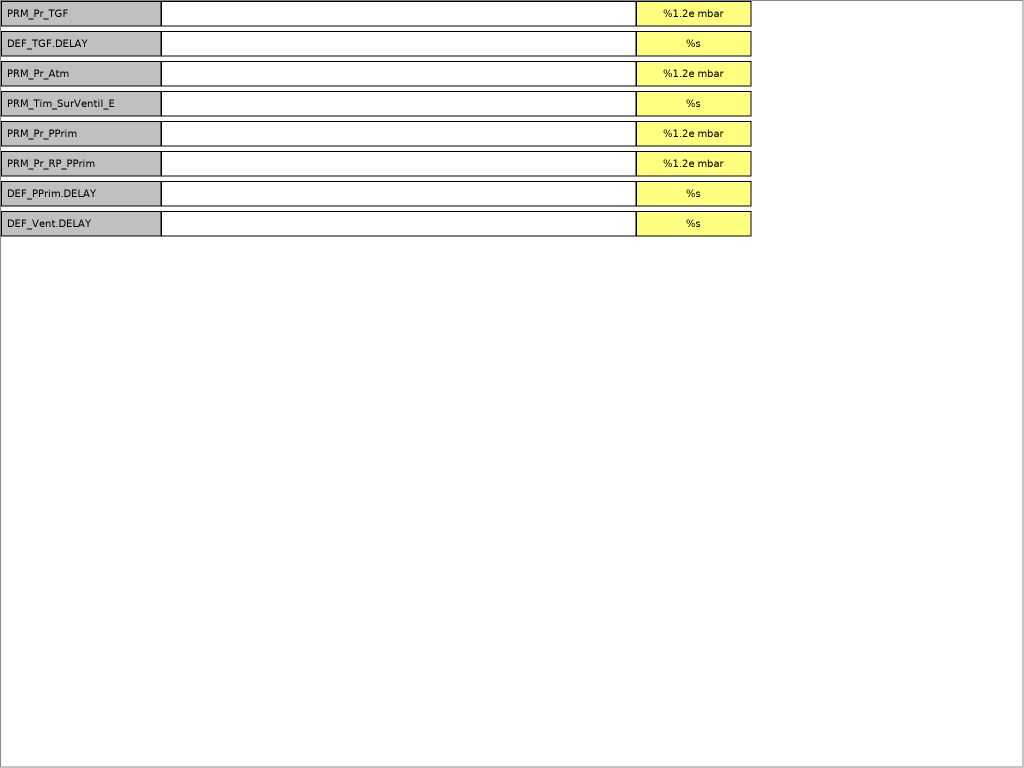
VISUALIZATION VISU_CONFIG_POMPAGE_SAS  // 1024x768
VAR_IN_OUT
	m_Input_PRG_POMPAGE : BLOCK_PRG_POMPAGE_SAS;
END_VAR
    Rectangle (161,1 475x25), text list: 'TextList_Config_Pompage', text index: 2
    Rectangle (636,1 115x25), "%1.2e mbar", text variable: m_Input_PRG_POMPAGE.POMPAGE.PRM_Pr_TGF, input disabled if: NOT Global_Variables.PRG_USER.ACTU_USER.CONF_MACHINE
        OnMouseClick: write the text variable via VisuDialogs.NumpadExtended, min 10, max 1000
    Rectangle (1,1 160x25), "PRM_Pr_TGF"
    Rectangle (161,31 475x25), text list: 'TextList_Config_Pompage', text index: 3
    Rectangle (636,31 115x25), "%s", text variable: m_Input_PRG_POMPAGE.POMPAGE.DEF_TGF.DELAY, input disabled if: NOT Global_Variables.PRG_USER.ACTU_USER.CONF_MACHINE
        OnMouseClick: write the text variable via VisuDialogs.Keypad
    Rectangle (1,31 160x25), "DEF_TGF.DELAY"
    Rectangle (161,61 475x25), text list: 'TextList_Config_Pompage', text index: 4
    Rectangle (161,91 475x25), text list: 'TextList_Config_Pompage', text index: 5
    Rectangle (636,61 115x25), "%1.2e mbar", text variable: m_Input_PRG_POMPAGE.POMPAGE.PRM_Pr_Atm, input disabled if: NOT Global_Variables.PRG_USER.ACTU_USER.CONF_MACHINE
        OnMouseClick: write the text variable via VisuDialogs.Numpad, min 100, max 1000
    Rectangle (1,61 160x25), "PRM_Pr_Atm"
    Rectangle (636,91 115x25), "%s", text variable: m_Input_PRG_POMPAGE.POMPAGE.PRM_Tim_SurVentil_E, input disabled if: NOT Global_Variables.PRG_USER.ACTU_USER.CONF_MACHINE
        OnMouseClick: write the text variable via VisuDialogs.Keypad
    Rectangle (1,91 160x25), "PRM_Tim_SurVentil_E"
    Rectangle (161,121 475x25), text list: 'TextList_Config_Pompage', text index: 6
    Rectangle (636,121 115x25), "%1.2e mbar", text variable: m_Input_PRG_POMPAGE.POMPAGE.PRM_Pr_PPrim, input disabled if: NOT Global_Variables.PRG_USER.ACTU_USER.CONF_MACHINE
        OnMouseClick: write the text variable via VisuDialogs.NumpadExtended, min 1e-3, max 1e-1
    Rectangle (1,121 160x25), "PRM_Pr_PPrim"
    Rectangle (1,151 160x25), "PRM_Pr_RP_PPrim"
    Rectangle (161,151 475x25), text list: 'TextList_Config_Pompage', text index: 7
    Rectangle (636,151 115x25), "%1.2e mbar", text variable: m_Input_PRG_POMPAGE.POMPAGE.PRM_Pr_RP_PPrim, input disabled if: NOT Global_Variables.PRG_USER.ACTU_USER.CONF_MACHINE
        OnMouseClick: write the text variable via VisuDialogs.NumpadExtended, min 1e-3, max 1e-1
    Rectangle (1,181 160x25), "DEF_PPrim.DELAY"
    Rectangle (161,181 475x25), text list: 'TextList_Config_Pompage', text index: 8
    Rectangle (636,181 115x25), "%s", text variable: m_Input_PRG_POMPAGE.POMPAGE.DEF_PPRIM.DELAY, input disabled if: NOT Global_Variables.PRG_USER.ACTU_USER.CONF_MACHINE
        OnMouseClick: write the text variable via VisuDialogs.Keypad
    Rectangle (1,211 160x25), "DEF_Vent.DELAY"
    Rectangle (161,211 475x25), text list: 'TextList_Config_Pompage', text index: 9
    Rectangle (636,211 115x25), "%s", text variable: m_Input_PRG_POMPAGE.POMPAGE.DEF_VENT.DELAY, input disabled if: NOT Global_Variables.PRG_USER.ACTU_USER.CONF_MACHINE
        OnMouseClick: write the text variable via VisuDialogs.Keypad
END_VISUALIZATION

(* stored: Version 1.1.0.1, ProductVersion 3.1.4024.10
   Visu VISU_CONFIG_POMPAGE_SAS: Id {415d8b29-1af9-4deb-a5d4-9765c2b5afb3} *)
